# EPICS autosave request: soft_iocs/meas_comp/iocBoot/iocmeas_comp/auto_settings.req
file "ETC_settings.req", P=18ID:ETC:
file "E1608_settings.req", P=18ID:E1608:
